Fanuc KAREL source: ka00027.KL

PROGRAM KA00027
%NOLOCKGROUP
VAR
SRC:BOOLEAN;DST:BOOLEAN
BEGIN
--
SRC=TRUE
DST=SRC
END KA00027
